TYPE ST_HMI_G120Ctrl :
STRUCT
	stRun				: ST_HMI_Buttons;
	stReset				: ST_HMI_Buttons;
	nSpeedHz 			: UINT;
	stInvertDirection	: ST_HMI_Buttons;
END_STRUCT
END_TYPE

(* stored: Version 1.1.0.1, ProductVersion 3.1.4024.15
   DUT ST_HMI_G120Ctrl: Id {82340275-35e2-4444-a46a-a7b70d601128} *)
